SUBAPPLICATION SoftKeySR_PC_A_OPC_Adapter (* Geraet A (Station 11, 192.168.1.11): wie SoftKeySR_PC_A_OPC, aber HMI (2 SoftKeys + GreenWhiteBackground) und OPC-UA-Trigger sind getrennt - SoftKeySR_ASR_AX buendelt die HMI hinter einem ASR_AX-Plug, ASR_AX_CLIENT_0_SUBSCRIBE_1 buendelt die 2 CLIENT_0-Instanzen + AX_SUBSCRIBE_1 hinter einem ASR_AX-Socket - 'SUB style': das Protokoll steckt im MyLib::sys-Composite, nicht in der Resource des Geraets *)
  (* Standard: 61499-2; Description: Copyright (c) 2026 Meisterschulen am Ostbahnhof This program and the accompanying materials are made available under the terms of the Eclipse Public License 2.0 which is available at https://www.eclipse.org/legal/epl-2.0/ SPDX-License-Identifier: EPL-2.0 *)
  (* Version 1.0, 2026-09-04, Franz Höpfinger, Meisterschulen am Ostbahnhof, initial API and implementation and/or initial documentation *)
  PACKAGE MyLib::sys;
  IMPORT isobus::UT::Q::const::IDs::ID_NULL;
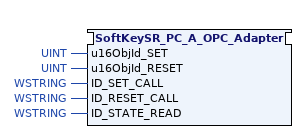
  VAR_INPUT
    u16ObjId_SET : UINT := ID_NULL; (* Object ID SoftKey Set (traegt auch das GreenWhiteBackground) *)
    u16ObjId_RESET : UINT := ID_NULL; (* Object ID SoftKey Reset *)
    ID_SET_CALL : WSTRING; (* Remote-Methodenadresse (ACTION=CALL_METHOD) fuer den Set-Methodenaufruf auf Geraet B *)
    ID_RESET_CALL : WSTRING; (* Remote-Methodenadresse (ACTION=CALL_METHOD) fuer den Reset-Methodenaufruf auf Geraet B *)
    ID_STATE_READ : WSTRING; (* Lokal ueberwachte Adresse (BOOL, ACTION=READ) fuer den Flipflop-Zustand, wird von Geraet B remote beschrieben *)
  END_VAR
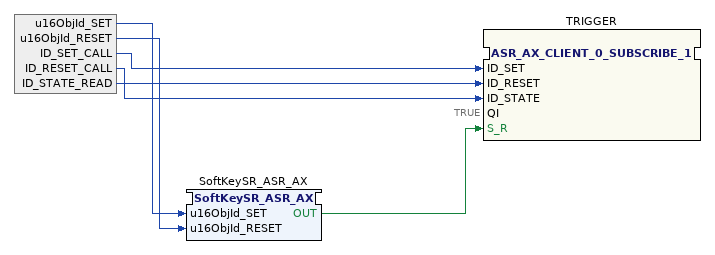
  FBS
    TRIGGER : adapter::net::ASR_AX_CLIENT_0_SUBSCRIBE_1(QI := TRUE);
  END_FBS
  SUBAPPS
    SoftKeySR_ASR_AX : MyLib::sys::SoftKeySR_ASR_AX;
  END_SUBAPPS
  DATA_CONNECTIONS
    ID_SET_CALL TO TRIGGER.ID_SET;
    ID_RESET_CALL TO TRIGGER.ID_RESET;
    ID_STATE_READ TO TRIGGER.ID_STATE;
    u16ObjId_SET TO SoftKeySR_ASR_AX.u16ObjId_SET;
    u16ObjId_RESET TO SoftKeySR_ASR_AX.u16ObjId_RESET;
  END_CONNECTIONS
  ADAPTER_CONNECTIONS
    SoftKeySR_ASR_AX.OUT TO TRIGGER.S_R;
  END_CONNECTIONS
END_SUBAPPLICATION
